// TIA Portal V19 export
DATA_BLOCK "DATA RECIEVED FROM MASTER DB"   // DB228
{ S7_Optimized_Access := 'FALSE' }
// stored: AutoNumber false
   VAR
      "REAL" : Real;
      REAL_1 : Real;
      REAL_2 : Real;
      REAL_3 : Real;
      REAL_4 : Real;
      REAL_5 : Real;
   END_VAR
BEGIN
END_DATA_BLOCK
